{attribute 'qualified_only'}
{attribute 'strict'}
{attribute 'to_string'}
TYPE E_Levi_States :
(
	LEVI_IDLE 						:= 0,
	LEVI_INIT 						:= 1,
	LEVI_READY 						:= 2,
	LEVI_PULLUP 					:= 3,
	LEVI_DROPDOWN 					:= 4,
	LEVI_LIFTOFF					:= 5,
	LEVI_LEVITATION					:= 6,
	LEVI_DESCEND					:= 7,
	LEVI_TESTING_INDIVIDUAL_DRIVES 	:= 8, 
	LEVI_ERROR						:= -1,
	LEVI_RESET_DRIVES				:= -2
) UINT;
END_TYPE

(* stored: Version 1.1.0.1
   DUT E_Levi_States: Id {4d8c88c9-363a-4885-aa20-1dd9d673ad95} *)
